PROGRAM prgPV
VAR
	fbPV						: FB_SunSpec_PV_Inverter_T;
	lrPowerPV					: LREAL;						//{#lynus.ag#()}
	byErrorWarningPV			: BYTE;							//{#lynus.ag#()}
END_VAR
VAR PERSISTENT
	lrCounterPV					: LREAL;						//{#lynus.ag#()}
END_VAR

// To-Do:
// adopt FB Declaration, change to correct FB
// adopt FB Definition, change to correct in/out Vars
// correct lrPowerPV definition
// correct lrCounterPV definition
// correct byErrorWarningPV definition

fbPV(
	bEnable:= TRUE, 
	sIPAdress:= '192.168.1.35', 
	byUnitID_Inverter:= 1, 
	stDataSunSpec=> , 
	stDataEMPower_PV=> , 
	stDataEMCounter_PV=> , 
	diNrOfEM_OUT_PV=> );

lrPowerPV := fbPV.stDataEMPower_PV.lrPowerTotal;
byErrorWarningPV := fbPV.stDataEMPower_PV.byErrorWarning;
	
IF fbPV.stDataEMCounter_PV.lrCounterEnergyT1_Production > lrCounterPV THEN  	
	lrCounterPV := fbPV.stDataEMCounter_PV.lrCounterEnergyT1_Production;
END_IF

END_PROGRAM

(* stored: Version 1.1.0.1, ProductVersion 3.1.4024.11
   POU prgPV: Id {52a4cf08-62d2-4b94-900b-2ea0759cae15}, SpecialFunc None *)
